% RSLogix 500 project FLIP-FLOP DEADZONE_BAK024.RSS, saved by version 10.00.00.00 %
PROJECT "UNTITLED"    % processor: Bul.1763 MicroLogix 1100 Series B %

PROGRAM FILES
  LAD 2   11 rungs

DATA FILES
  O0 OUTPUT  4 elements
  I1 INPUT  6 elements
  S2 STATUS  66 elements
  B3 BINARY  1 elements
  T4 TIMER  4 elements
  C5 COUNTER  1 elements
  R6 CONTROL  1 elements
  N7 INTEGER  4 elements
  F8 FLOAT  1 elements

LADDER 2
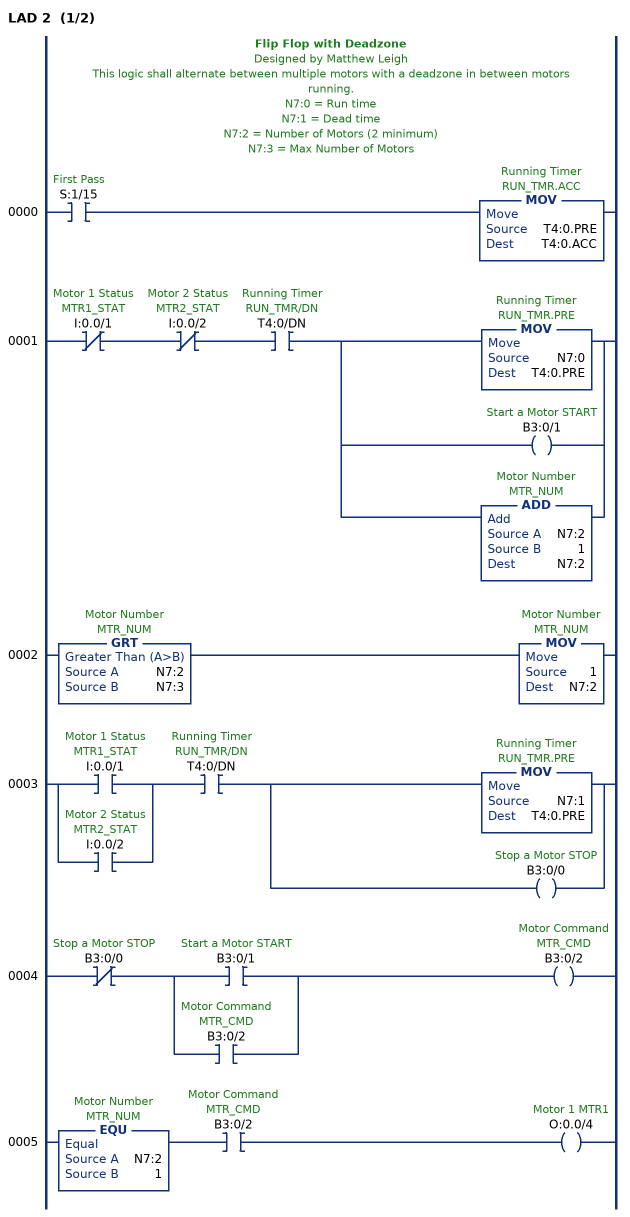
% Rung: 0 %
% TITLE: Flip Flop with Deadzone %
% Designed by Matthew Leigh
% 
% This logic shall alternate between multiple motors with a deadzone in between motors running.
%      N7:0 = Run time
%      N7:1 = Dead time
%      N7:2 = Number of Motors (2 minimum)
%      N7:3 = Max Number of Motors %
SOR XIC S:1/15 MOV T4:0.PRE T4:0.ACC EOR
%   S:1/15  "First Pass" %
%   T4:0  RUN_TMR  "Running Timer" %
% Rung: 1 %
SOR XIO I:0.0/1 XIO I:0.0/2 XIC T4:0/DN BST MOV N7:0 T4:0.PRE NXB OTE B3:0/1 NXB ADD N7:2 1 N7:2 BND EOR
%   I:0.0/1  MTR1_STAT  "Motor 1 Status" %
%   I:0.0/2  MTR2_STAT  "Motor 2 Status" %
%   T4:0  RUN_TMR  "Running Timer" %
%   N7:0  RUN_TM  "Running Time" %
%   B3:0/1  START  "Start a Motor" %
%   N7:2  MTR_NUM  "Motor Number" %
% Rung: 2 %
SOR GRT N7:2 N7:3 MOV 1 N7:2 EOR
%   N7:2  MTR_NUM  "Motor Number" %
%   N7:3  MAX_NUM  "Max Number of Motors" %
% Rung: 3 %
SOR BST XIC I:0.0/1 NXB XIC I:0.0/2 BND XIC T4:0/DN BST MOV N7:1 T4:0.PRE NXB OTE B3:0/0 BND EOR
%   I:0.0/1  MTR1_STAT  "Motor 1 Status" %
%   I:0.0/2  MTR2_STAT  "Motor 2 Status" %
%   T4:0  RUN_TMR  "Running Timer" %
%   N7:1  PAS_TM  "Pause Time" %
%   B3:0/0  STOP  "Stop a Motor" %
% Rung: 4 %
SOR XIO B3:0/0 BST XIC B3:0/1 NXB XIC B3:0/2 BND OTE B3:0/2 EOR
%   B3:0/0  STOP  "Stop a Motor" %
%   B3:0/1  START  "Start a Motor" %
%   B3:0/2  MTR_CMD  "Motor Command" %
% Rung: 5 %
SOR EQU N7:2 1 XIC B3:0/2 OTE O:0.0/4 EOR
%   N7:2  MTR_NUM  "Motor Number" %
%   B3:0/2  MTR_CMD  "Motor Command" %
%   O:0.0/4  MTR1  "Motor 1" %

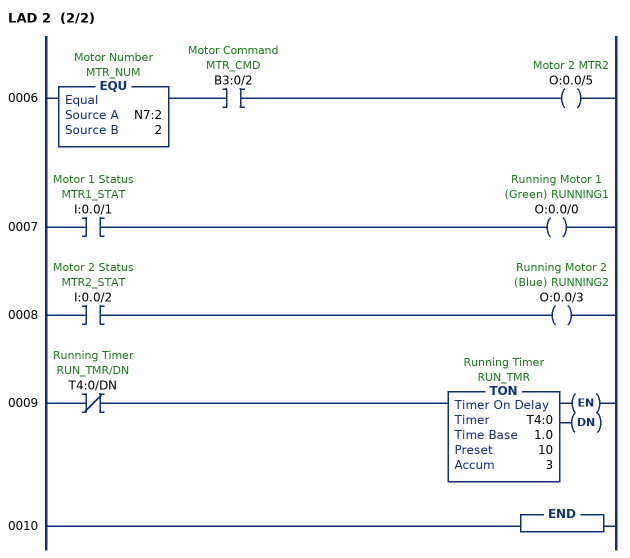
% Rung: 6 %
SOR EQU N7:2 2 XIC B3:0/2 OTE O:0.0/5 EOR
%   N7:2  MTR_NUM  "Motor Number" %
%   B3:0/2  MTR_CMD  "Motor Command" %
%   O:0.0/5  MTR2  "Motor 2" %
% Rung: 7 %
SOR XIC I:0.0/1 OTE O:0.0/0 EOR
%   I:0.0/1  MTR1_STAT  "Motor 1 Status" %
%   O:0.0/0  RUNNING1  "Running Motor 1 (Green)" %
% Rung: 8 %
SOR XIC I:0.0/2 OTE O:0.0/3 EOR
%   I:0.0/2  MTR2_STAT  "Motor 2 Status" %
%   O:0.0/3  RUNNING2  "Running Motor 2 (Blue)" %
% Rung: 9 %
SOR XIO T4:0/DN TON T4:0 1.0 10 3 EOR
%   T4:0  RUN_TMR  "Running Timer" %
% Rung: 10 %
SOR END EOR

OTHER DOCUMENTED ADDRESSES
  I:0  I
  T4:1  REV_TMR  "Reverse Timer"

DATA TABLE (non-zero values as saved)
DATA B3
% B3:0 % 0X0004
DATA T4
% .PRE .ACC %
% T4:0 % 10 3
% T4:1 % 6 0
% T4:3 % 3 0
DATA N7
% N7:0 % 10 5 1 2
